FUNCTION Convert_DINT_TO_DINT : BOOL
VAR_INPUT
	in : DINT;
	out : REFERENCE TO DINT;
END_VAR

out := in;
Convert_DINT_TO_DINT := TRUE;

END_FUNCTION

(* stored: Version 1.1.0.1, ProductVersion 3.1.4024.12
   POU Convert_DINT_TO_DINT: Id {1ecf48fd-15f8-4522-87b1-9c1347629742}, SpecialFunc None *)
